# EPICS autosave request: terminalServerApp/Db/acs_channel_settings.req
$(P)$(R):$(CHAN):APPLICATIONCFG.VAL
$(P)$(R):$(CHAN):PORTCFG.VAL
$(P)$(R):$(CHAN):ALIASCFG.VAL
$(P)$(R):$(CHAN):BAUDRATECFG.VAL
$(P)$(R):$(CHAN):DATABITSCFG.VAL
$(P)$(R):$(CHAN):STOPBITSCFG.VAL
$(P)$(R):$(CHAN):PARITYCFG.VAL
$(P)$(R):$(CHAN):FLOWCONTROLCFG.VAL
